FUNCTION_BLOCK integrator_1 (* Basic FB with empty ECC *)
  (* Standard: 61499-2 *)
  (* Version 1.0, 2021-05-19, Lenovo *)
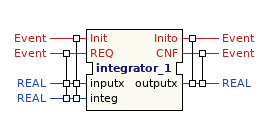
  EVENT_INPUT
    Init WITH inputx, integ;
    REQ WITH inputx, integ;
  END_EVENT
  EVENT_OUTPUT
    Inito WITH outputx;
    CNF WITH outputx;
  END_EVENT
  VAR_INPUT
    inputx : REAL;
    integ : REAL;
  END_VAR
  VAR_OUTPUT
    outputx : REAL;
  END_VAR
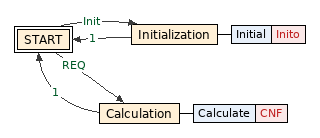
  EC_STATES
    START; (* Initial State *)
    Initialization : Initial -> Inito;
    Calculation : Calculate -> CNF;
  END_STATES
  EC_TRANSITIONS
    START TO Initialization := Init;
    Initialization TO START := 1;
    START TO Calculation := REQ;
    Calculation TO START := 1;
  END_TRANSITIONS
  ALGORITHM Initial IN ST: (* New Algorithm *)

  END_ALGORITHM
  ALGORITHM Calculate IN ST: (* New Algorithm *)
outputx:=(inputx*5)+integ;
  END_ALGORITHM
END_FUNCTION_BLOCK
